FUNCTION_BLOCK MECHC_VIEW (* View of a Linear Mechanism with Clamping *)
  (* Standard: 61499-1; Classification: View *)
  (* Version 0.2, 2004-10-07, JHC, Rockwell Automation, Added CNV input. *)
  (* Version 0.1, 2004-09-27, JHC, Rockwell Automation, Moved CLAMP after WKPC for consistency with MECH_VIEW. *)
  (* Version 0.0, 2002-05-21, JHC, Rockwell Automation, Copied/Modified from MECH_VIEW. *)
  (* Compiler header: package fb.rt.mva; *)
  (* Compiler classdef: public class MECHC_VIEW extends MECH_VIEW *)
  (* Compiler Java Sun JDK 1.4.2 *)
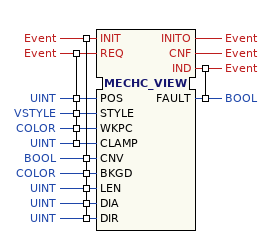
  EVENT_INPUT
    INIT WITH BKGD, LEN, DIA, DIR, CNV; (* Initialize *)
    REQ WITH POS, CLAMP, STYLE, WKPC; (* Update the display *)
  END_EVENT
  EVENT_OUTPUT
    INITO; (* Initialized *)
    CNF; (* Display Updated *)
    IND WITH FAULT; (* Change in FAULT status *)
  END_EVENT
  VAR_INPUT
    POS : UINT; (* Mechanism displacement,% *)
    STYLE : VSTYLE := RING; (* View style *)
    WKPC : COLOR := blue; (* Foreground Color *)
    CLAMP : UINT; (* Clamp or gate position,% *)
    CNV : BOOL; (* 0=Paint workpiece with clamp,1=Paint as conveyor with gate at end. *)
    BKGD : COLOR := blue; (* Background Color *)
    LEN : UINT; (* Length in Diameters *)
    DIA : UINT; (* Diameter *)
    DIR : UINT; (* Orientation:0=L/R,1=T/B,2=R/L,3=B/T *)
  END_VAR
  VAR_OUTPUT
    FAULT : BOOL; (* 0=Normal,1=Fault *)
  END_VAR
END_FUNCTION_BLOCK
